FUNCTION_BLOCK EdgeDetector_1
VAR_INPUT
	inputValue : BOOL ;
END_VAR

VAR_OUTPUT
	riesingEdge :BOOL;
	fallingEdge :BOOL;
END_VAR
VAR
	safeStatus:BOOL;
	totzeit : INT;
END_VAR

fallingEdge := FALSE;
riesingEdge := FALSE;
IF totzeit <1 THEN
	IF safeStatus = FALSE AND inputValue = TRUE THEN
		riesingEdge:= TRUE;
		totzeit := 100;
	ELSIF safeStatus = TRUE AND inputValue = FALSE THEN
		fallingEdge:= TRUE;
		totzeit := 100;
	END_IF
	ELSE
	totzeit := totzeit -1;
END_IF
safeStatus := inputValue;

END_FUNCTION_BLOCK

(* stored: Version 1.1.0.1, ProductVersion 3.1.4022.12
   POU EdgeDetector_1: Id {20a7cb78-1e55-4a66-9642-d8d122f25561}, SpecialFunc None *)
